TYPE ST_AutoAddsBoxesStatus EXTENDS ST_StatusBasic :
STRUCT
	InterventionRequest	 : BOOL;
	FeedingBoxes		 :BOOL;
END_STRUCT
END_TYPE

(* stored: Version 1.1.0.1, ProductVersion 3.1.4024.13
   DUT ST_AutoAddsBoxesStatus: Id {7c508ce6-1e40-438c-b5a8-982209b43ba2} *)
